Fanuc KAREL source: kt00507.KL

PROGRAM KT00507
%STACKSIZE=65535
%PRIORITY=65535
%NOLOCKGROUP
VAR
P1 : XYZWPR
P2 : XYZWPREXT
OUT : JOINTPOS9
BEGIN
P1.X=1.0
P2.Y=2.0
-- UNRESOLVED_PC line 10 opcodes [49 7E 49 7E 60 7E 4A] marker_code=40
END KT00507
